FUNCTION_BLOCK COARSE_MOVE_V2 (* Basic Function Block Type *)
  (* Standard: 61499-2 *)
  (* Version 0.0, 4/28/2023, Dmitrii, Flexbridge AB, Template *)
  PACKAGE UAO.Hackathon;
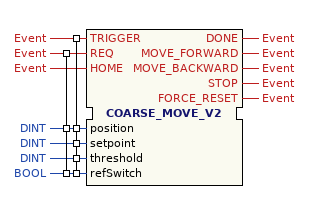
  EVENT_INPUT
    TRIGGER WITH setpoint, threshold, position, refSwitch; (* Normal Execution Request *)
    REQ WITH position, refSwitch;
    HOME;
  END_EVENT
  EVENT_OUTPUT
    DONE; (* Execution Confirmation *)
    MOVE_FORWARD;
    MOVE_BACKWARD;
    STOP;
    FORCE_RESET; (* Force position monitor reset *)
  END_EVENT
  VAR_INPUT
    position : DINT;
    setpoint : DINT;
    threshold : DINT;
    refSwitch : BOOL;
  END_VAR
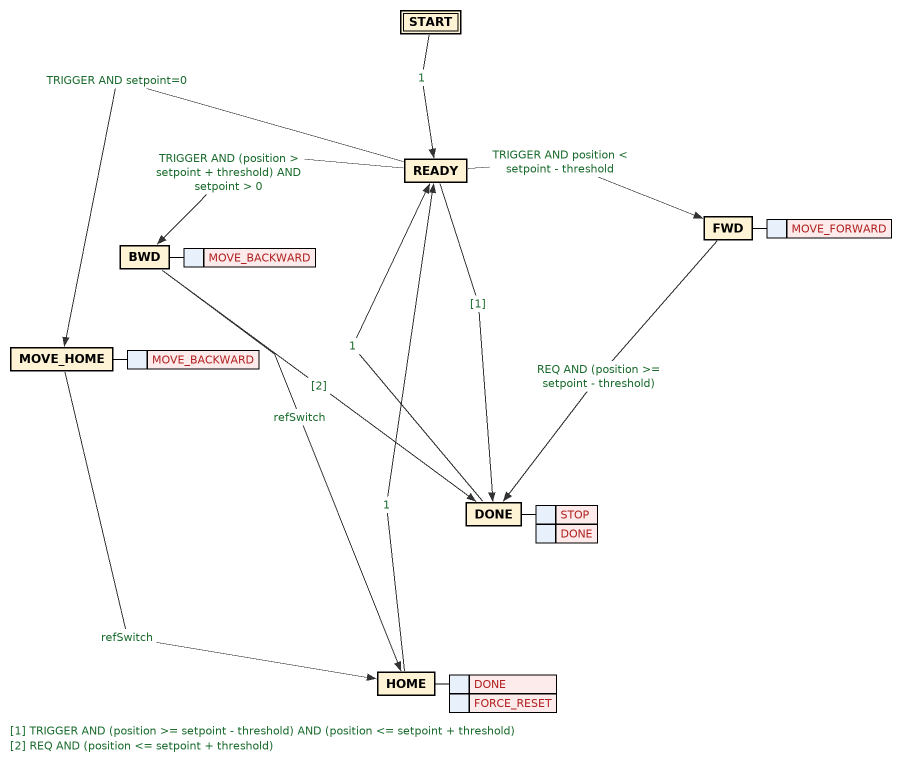
  EC_STATES
    START; (* Initial State *)
    READY;
    FWD : -> MOVE_FORWARD;
    BWD : -> MOVE_BACKWARD;
    DONE : -> STOP, -> DONE;
    HOME : -> DONE, -> FORCE_RESET;
    MOVE_HOME : -> MOVE_BACKWARD;
  END_STATES
  EC_TRANSITIONS
    MOVE_HOME TO HOME := refSwitch;
    START TO READY := 1;
    READY TO FWD := TRIGGER AND position < setpoint - threshold;
    FWD TO DONE := REQ AND (position >= setpoint - threshold);
    DONE TO READY := 1;
    READY TO BWD := TRIGGER AND (position > setpoint + threshold) AND setpoint > 0;
    BWD TO DONE := REQ AND (position <= setpoint + threshold);
    READY TO DONE := TRIGGER AND (position >= setpoint - threshold) AND (position <= setpoint + threshold);
    BWD TO HOME := refSwitch;
    HOME TO READY := 1;
    READY TO MOVE_HOME := TRIGGER AND setpoint=0;
  END_TRANSITIONS
  ALGORITHM INIT IN ST: (* Initialization algorithm *)
;
  END_ALGORITHM
  ALGORITHM REQ IN ST: (* Normally executed algorithm *)
;
  END_ALGORITHM
END_FUNCTION_BLOCK
